FUNCTION_BLOCK DamperModule
VAR_INPUT
	EN: BOOL;
	UnitID: BYTE;
	ModbusTCP: REFERENCE TO Modbus;
	Exercise: BOOL;
	ResetSmokeDetector: bool;
	SxDuoCommand: SxDuoCommand;
	{attribute 'TcEncoding':='UTF-8'}
	WriteText: STRING;
END_VAR
VAR_OUTPUT
	ENO: BOOL;
	Error: BOOL;
	Fire: BOOL;
	Exercising: BOOL;
	DamperError: BOOL;
	ServiceAlarm: BOOL;
	{attribute 'TcEncoding':='UTF-8'}
	Text: STRING;
	SxDuoStatus: SxDuoStatus;
END_VAR
VAR
	ModbusReadBits3: ModbusReadBits;
	ModbusWriteBits3: ModbusWriteBits;
	ModbusReadWordArray_0: ModbusReadWordArray;
END_VAR
VAR // added by the converter: edge detectors and wires of the graphical bodies
    _s1 : SxDuoStatus;
    _w1, _w2 : ANY;
END_VAR


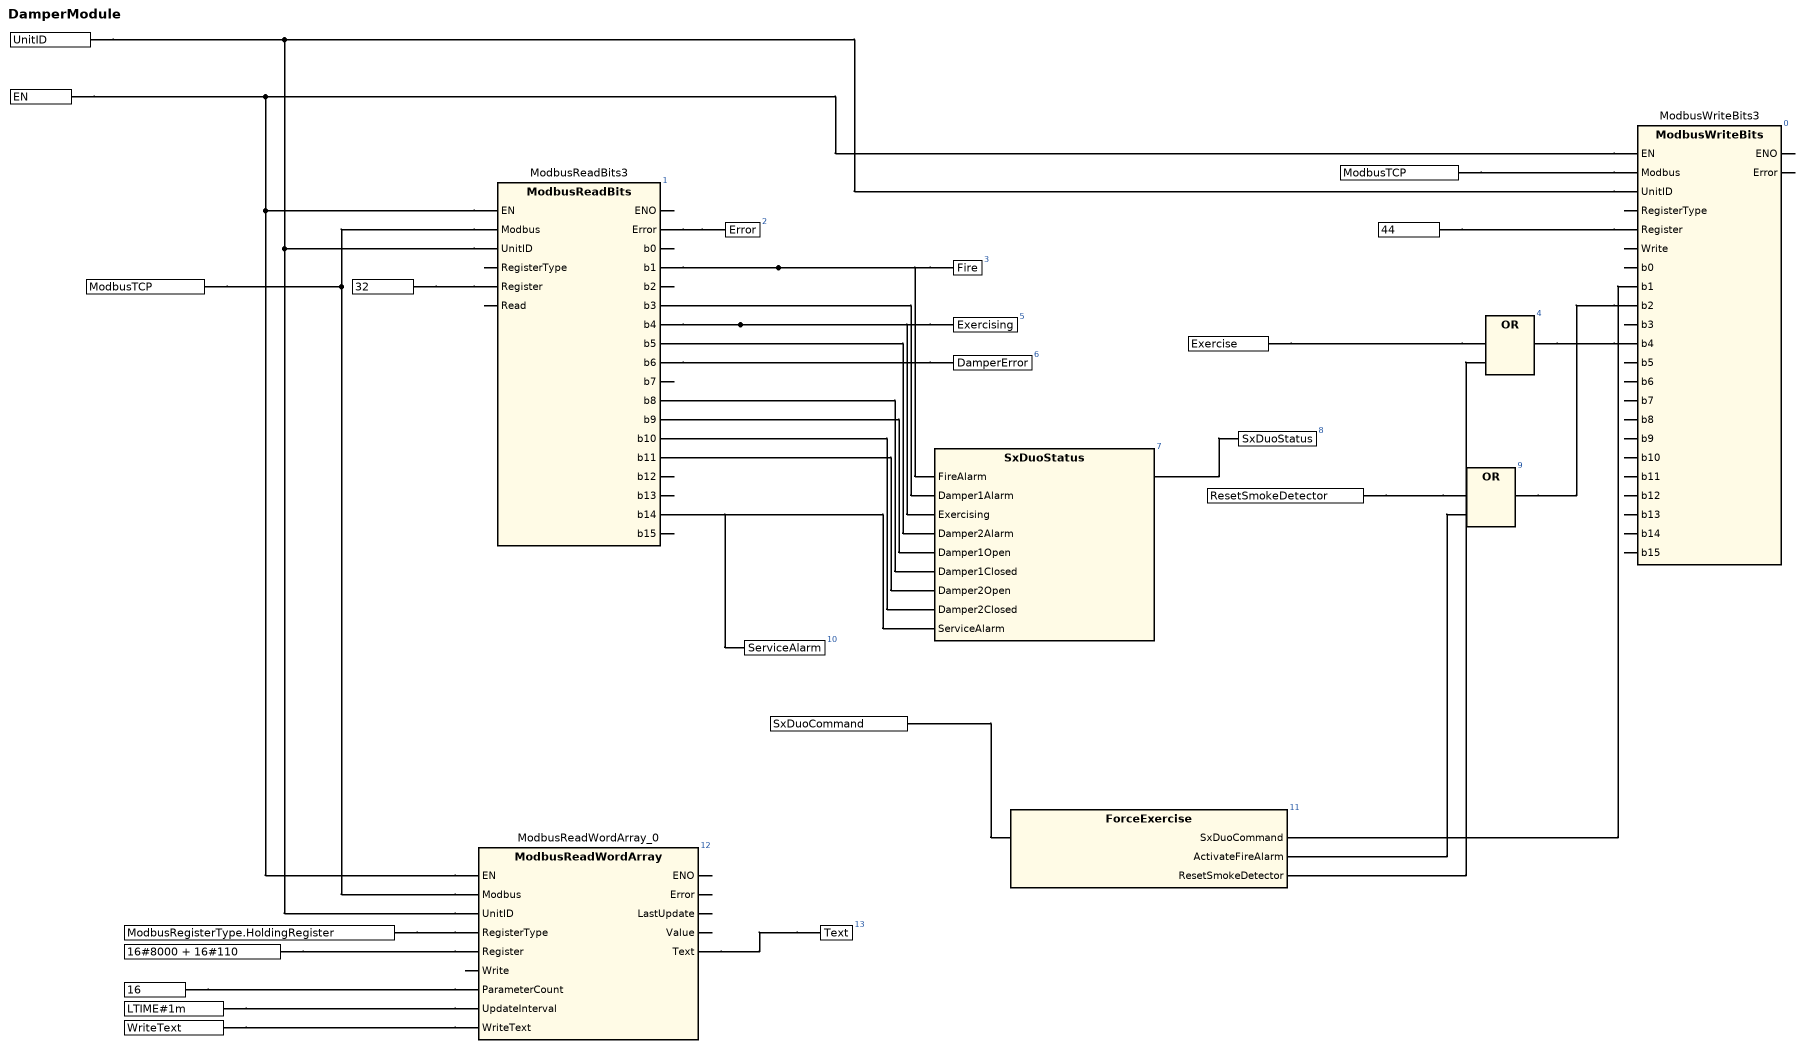
// PAGE
ModbusWriteBits3(
    EN := EN,
    Modbus := ModbusTCP,
    UnitID := UnitID,
    Register := 44,
    b1 := ???,
    b2 := _w1,
    b4 := _w2); // ModbusWriteBits
ModbusReadBits3(EN := EN, Modbus := ModbusTCP, UnitID := UnitID, Register := 32); // ModbusReadBits
Error := ModbusReadBits3.Error;
Fire := ModbusReadBits3.b1;
_w2 := Exercise OR ???;
Exercising := ModbusReadBits3.b4;
DamperError := ModbusReadBits3.b6;
// compose _s1 : SxDuoStatus
_s1.FireAlarm := ModbusReadBits3.b1;
_s1.Damper1Alarm := ModbusReadBits3.b3;
_s1.Exercising := ModbusReadBits3.b4;
_s1.Damper2Alarm := ModbusReadBits3.b5;
_s1.Damper1Open := ModbusReadBits3.b9;
_s1.Damper1Closed := ModbusReadBits3.b8;
_s1.Damper2Open := ModbusReadBits3.b11;
_s1.Damper2Closed := ModbusReadBits3.b10;
_s1.ServiceAlarm := ModbusReadBits3.b14;
SxDuoStatus := _s1;
_w1 := ResetSmokeDetector OR ???;
ServiceAlarm := ModbusReadBits3.b14;
ModbusReadWordArray_0(
    EN := EN,
    Modbus := ModbusTCP,
    UnitID := UnitID,
    RegisterType := ModbusRegisterType.HoldingRegister,
    Register := 16#8000 + 16#110,
    ParameterCount := 16,
    UpdateInterval := LTIME#1m,
    WriteText := WriteText); // ModbusReadWordArray
Text := ModbusReadWordArray_0.Text;

METHOD StartWrite : BOOL
VAR_INPUT
END_VAR
ModbusWriteBits3.EN := TRUE;
END_METHOD

END_FUNCTION_BLOCK

(* stored: Version 1.1.0.1, ProductVersion 3.1.4024.6
   POU DamperModule: Id {164cac92-565a-49e6-ae1e-a498db03c341}, SpecialFunc None
   Method StartWrite: Id {12cbacf6-2bb7-4d6a-9031-5da0b128d7b9} *)
